// TIA Portal V15.1 export
// export: Created 2024-06-21T08:40:36.5097904Z, ExportSetting WithDefaults, DisplayName Totally Integrated Automation Portal, DisplayVersion V15.1 Update 5, DisplayName TIA Portal Openness, DisplayVersion V15.1 Update 5, DisplayName SINAMICS Startdrive Advanced, DisplayVersion V15.1, DisplayName G130, G150, S120, S150, SINAMICS MV, S210, DisplayVersion V15.1, DisplayName G110M, G120, G120C, G120D, G120P, DisplayVersion V15.1, DisplayName STEP 7 Professional, DisplayVersion V15.1 Update 5, DisplayName STEP 7 Safety, DisplayVersion V15.1, DisplayName WinCC Professional, DisplayVersion V15.1 Update 5, DisplayName SIMATIC Visualization Architect, DisplayVersion V15.1
ORGANIZATION_BLOCK "RACK_FLT"   // OB86, FBD, RackOrStationFailure
TITLE = RACK_FLT
{ S7_Optimized_Access := 'TRUE' }
AUTHOR : VCC
VERSION : 0.0.0.0
// =============================================================================
// Loss Of Rack Fault
// =============================================================================
// stored: IsIECCheckEnabled false, SetENOAutomatically False
   VAR_INPUT
      LADDR : HW_IO;   // Hardware identifier
      Event_Class : Byte;   // Event class
      Fault_ID : Byte;   // Fault identifier
   END_VAR
   VAR_TEMP
      OB86_RACKS_FLTD : Array[0..31] of Bool;
      OB86_DATE_TIME : Date_And_Time;   // Date and time OB86 started
   END_VAR
BEGIN

REGION Network 1: **** 1 - Inputs **** Incrementation of number of executions
   // Incrementation of number of executions
   // If first bit in local data is set then there is a rack fault, if not set then 
   // the rack comes back online, so incrementation is not neccessary if the bit is 
   // not set (prevents alarm from coming up)
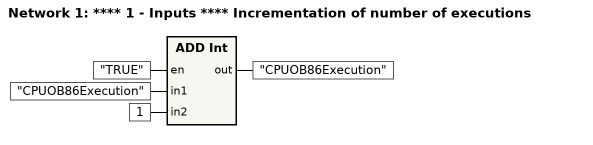
   IF "TRUE" THEN "CPUOB86Execution" := "CPUOB86Execution" + 1; END_IF;
END_REGION
END_ORGANIZATION_BLOCK
